// TIA Portal V16 export
// export: Created 2022-11-14T17:35:50.519923Z, ExportSetting WithDefaults, DisplayName Totally Integrated Automation Portal, DisplayVersion V16, DisplayName TIA Portal Version Control Interface, DisplayVersion V16, DisplayName TIA Portal Openness, DisplayVersion V16, DisplayName STEP 7 Professional, DisplayVersion V16, DisplayName STEP 7 Safety, DisplayVersion V16, DisplayName WinCC Advanced, DisplayVersion V16
DATA_BLOCK "DB320_PID"   // DB320
TITLE = PID
{ S7_Optimized_Access := 'FALSE' }
VERSION : 0.1
// stored: AutoNumber false, IsOnlyStoredInLoadMemory false, IsWriteProtectedInAS false
   VAR RETAIN
      PID { S7_SetPoint := 'True'} : "PID";
   END_VAR
BEGIN
   PID.proporzionale := 0;
   PID.integrativo := 0;
   PID.segnale := 0;
   PID.maxSegnale := 1000;
   PID.minSegnale := 0;
   PID.setPointShow := 265;
   PID.tiro := 0;
   PID.vParP := 70;
   PID.vParI := 70;
   PID.svuota := TRUE;
   PID.attiva := TRUE;
   PID.setTiro := FALSE;
   PID."timer" := T#0MS;
END_DATA_BLOCK
